// TIA Portal V18 export
TYPE "RCS_typeAteqF620Visual"
   STRUCT
      Trigger : Struct
         SetProg : Bool;
         Measure : Bool;
      END_STRUCT;
      Set : Struct
         ProgNo : UInt;   // document name
      END_STRUCT;
      Status { ExternalWritable := 'False'} : Struct
         InstanceName : WString[20];
         DeviceReady : Bool;
         Ready : Bool;
         Error : Bool;
         SetProgOk : Bool;
         MeasureOk : Bool;
         ErrorCode : UInt;
         Result : Struct
            PassPart : Bool;
            FailTestPart : Bool;
            FailRefPart : Bool;
            Alarm : Bool;
            PressureError : Bool;
            PartRecoverable : Bool;
            CalibError : Bool;
            CalibCheckError : Bool;
            AtrFault : Bool;
            Leak : Struct
               Value : Real;
               Unit : String[10];
            END_STRUCT;
         END_STRUCT;
         Pressure : Struct
            Value : Real;
            Unit : String[10];
         END_STRUCT;
         ActProgStep : UInt;
         ActProgNo : UInt;
         ElapsedTime : Time;
      END_STRUCT;
   END_STRUCT;
END_TYPE
